VISUALIZATION VISU_AutoCycle  // 800x480
END_VISUALIZATION

(* stored: Version 1.1.0.1, ProductVersion 3.1.4026.18
   Visu VISU_AutoCycle: Id {100b862d-9fd7-41cb-a4b7-c58e6cf2b5a6} *)
